(* Schneider Machine Expert - Basic project Questao3.6_FelipeV1_20241010, file version 2.9.0.0 *)
(* ProjectInformations: Name=Novo projeto *)

HARDWARE
  Cpu 0: TM221M16R/G
  EthernetConfiguration: NetworkName=M221, IpAllocationMode=FixedAddress, IpAddress=0.0.0.0, SubnetMask=0.0.0.0
  SerialLineConfiguration: Baud=Baud19200, Parity=ParityEven, DataBits=DataBits8, StopBits=StopBits1, PhysicalMedium=PhysicalMediumRs485, TransmissionMode=TransmissionModeModbusRtu, SlaveId=1, Addressing=SlaveAddressing
  MastTask: UsePeriodScanMode=false, PeriodScan=100
  FastTask: Period=255
  CpuBehavior: StartingMode=StartAsPreviousState, AutoSaveRamOnEeprom=true, WatchdogPeriod=250

SYMBOLS  (address, symbol, comment, settings)
  %M0       ACIO_GAT_G
  %M5       CONT_A_LIGA
  %M6       CONT_A_DESL
  %M7       CONT_E_LIGA
  %M8       CONT_E_DESL
  %M20      FT_TEMP2
  %TM0      TEMP_LIG  [Preset=5, Base=OneSecond]
  %TM1      TEMP_DESL  [Preset=5, Base=OneSecond]
  %I0.0     GAT_G
  %Q0.0     ACIO_CON_A
  %Q0.1     ACIO_RELE_E

POU Entradas
  (* SectionNumber=1 *)

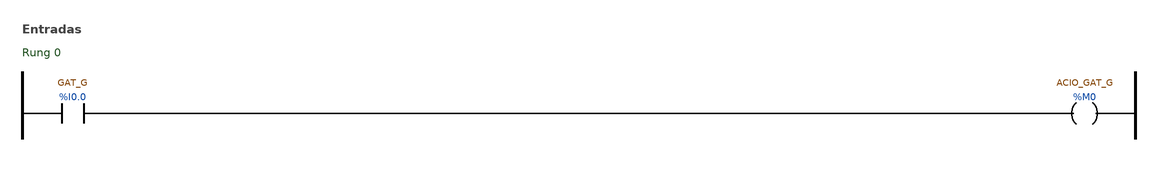

// Rung 0
  LD %I0.0                (* GAT_G *)
  ST %M0                  (* ACIO_GAT_G *)
  // as ST:
  //   ACIO_GAT_G := GAT_G;

POU Lógica
  (* SectionNumber=2 *)

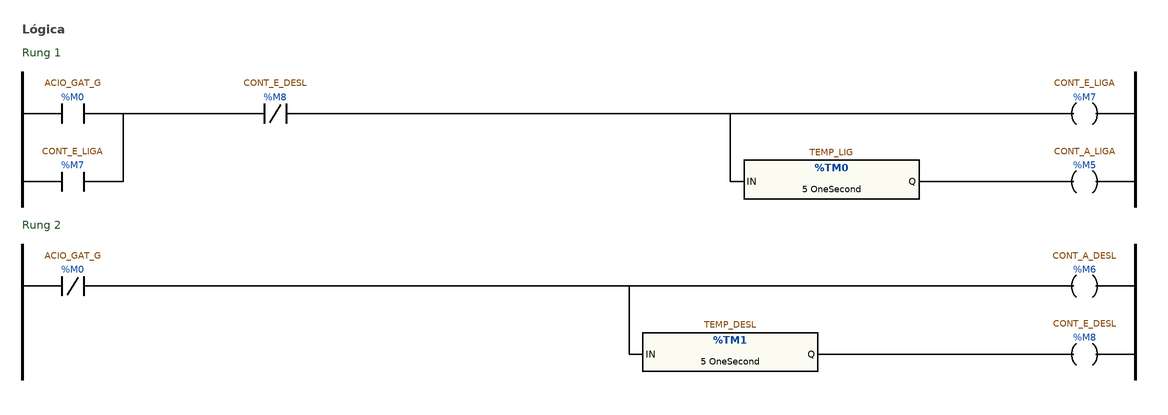

// Rung 1
  LD 1
  MULTIFB
  LD 1
  AND %M0                 (* ACIO_GAT_G *)
  OR %M7                  (* CONT_E_LIGA *)
  ANDN %M8                (* CONT_E_DESL *)
  ST %MW2009:X0
  LD %MW2009:X0
  ST %M7                  (* CONT_E_LIGA *)
  BLK %TM0                (* TEMP_LIG *)
  LD %MW2009:X0
  IN
  OUT_BLK
  LD Q
  ST %M5                  (* CONT_A_LIGA *)
  END_BLK
  MULTIFB
  // as ST:
  //   _t1 := (ACIO_GAT_G OR CONT_E_LIGA) AND NOT CONT_E_DESL;
  //   CONT_E_LIGA := _t1;
  //   TEMP_LIG(IN := _t1);
  //   CONT_A_LIGA := TEMP_LIG.Q;

// Rung 2
  LD 1
  MULTIFB
  LD 1
  ANDN %M0                (* ACIO_GAT_G *)
  ST %MW2009:X0
  LD %MW2009:X0
  ST %M6                  (* CONT_A_DESL *)
  BLK %TM1                (* TEMP_DESL *)
  LD %MW2009:X0
  IN
  OUT_BLK
  LD Q
  ST %M8                  (* CONT_E_DESL *)
  END_BLK
  MULTIFB
  // as ST:
  //   CONT_A_DESL := NOT ACIO_GAT_G;
  //   TEMP_DESL(IN := NOT ACIO_GAT_G);
  //   CONT_E_DESL := TEMP_DESL.Q;

POU Saídas
  (* SectionNumber=3 *)

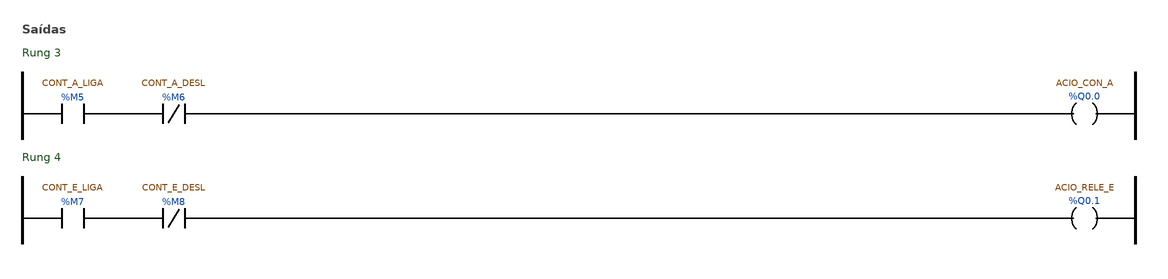

// Rung 3
  LD %M5                  (* CONT_A_LIGA *)
  ANDN %M6                (* CONT_A_DESL *)
  ST %Q0.0                (* ACIO_CON_A *)
  // as ST:
  //   ACIO_CON_A := CONT_A_LIGA AND NOT CONT_A_DESL;

// Rung 4
  LD %M7                  (* CONT_E_LIGA *)
  ANDN %M8                (* CONT_E_DESL *)
  ST %Q0.1                (* ACIO_RELE_E *)
  // as ST:
  //   ACIO_RELE_E := CONT_E_LIGA AND NOT CONT_E_DESL;
